PROGRAM MAIN
VAR_OUTPUT
	localTime : TIMESTRUCT;
END_VAR
VAR
	execute AT %I* : BOOL;
	trigger : R_TRIG;
	
	newBundle AT %M* : Bundle;
	newBundleConveyorsOccupied : ARRAY[1..6] OF BOOL;
	bundlesQueue : ARRAY[0..CONSTS.maxQueue] OF Bundle;
	numBundles : INT;
	
	buffers : ARRAY[1..CONSTS.numBuffers] OF IndexedBuffer;
END_VAR
VAR //transfer junctions are clear
	transferJunctionClear_A4 AT %I* : BOOL;
	transferJunctionClear_A5 AT %I* : BOOL;
	transferJunctionClear_A2 AT %I* : BOOL;
END_VAR
VAR CONSTANT //area 3 indexes for the transfer junctions
	transferJunctionIndex_A4 : INT := 5;
	transferJunctionIndex_A5 : INT := 10;
	transferJunctionIndex_A2 : INT := 20;
END_VAR

(*
Area 3 contains <n> buffers, each index contains 6 conveyors
	this allows each buffer to carry up to a theoretical maximum of 6 bundles - realistically this will be limited to 3

implementation:
	each buffer stores 6 iterators (1 for each conveyor) to point to an element in bundlesQueue, and a master conveyor mode request
	set the requested mode for all conveyors within a buffer to the highest priority request
	then use an external module calculate the links and set the modes
	
on receipt of new bundle:
	add to bundle queue
	identify which conveyor lines the bundle sits on
*)

initialize();
callBuffers();

METHOD PRIVATE blocks : BOOL
VAR_INPUT
END_VAR
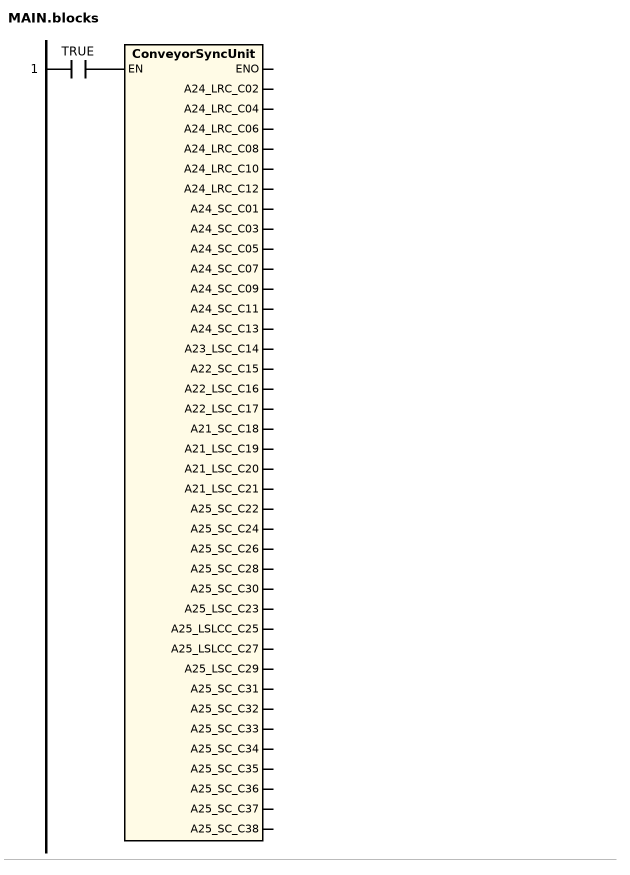
// NETWORK 1
ConveyorSyncUnit();
END_METHOD

METHOD callBuffers : BOOL
VAR_INPUT
END_VAR
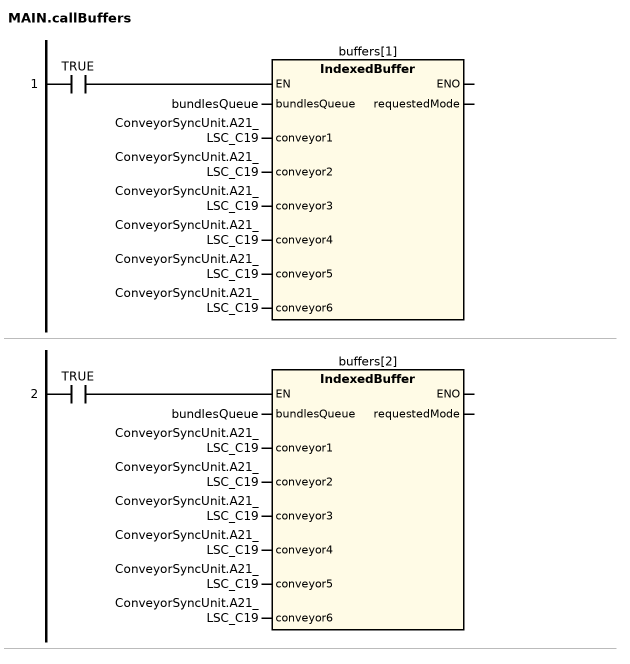
// NETWORK 1
buffers[1](
    bundlesQueue := bundlesQueue,
    conveyor1 := ConveyorSyncUnit.A21_LSC_C19,
    conveyor2 := ConveyorSyncUnit.A21_LSC_C19,
    conveyor3 := ConveyorSyncUnit.A21_LSC_C19,
    conveyor4 := ConveyorSyncUnit.A21_LSC_C19,
    conveyor5 := ConveyorSyncUnit.A21_LSC_C19,
    conveyor6 := ConveyorSyncUnit.A21_LSC_C19); // IndexedBuffer

// NETWORK 2
buffers[2](
    bundlesQueue := bundlesQueue,
    conveyor1 := ConveyorSyncUnit.A21_LSC_C19,
    conveyor2 := ConveyorSyncUnit.A21_LSC_C19,
    conveyor3 := ConveyorSyncUnit.A21_LSC_C19,
    conveyor4 := ConveyorSyncUnit.A21_LSC_C19,
    conveyor5 := ConveyorSyncUnit.A21_LSC_C19,
    conveyor6 := ConveyorSyncUnit.A21_LSC_C19); // IndexedBuffer
END_METHOD

METHOD PRIVATE handleJunctions : BOOL
VAR_INPUT
END_VAR
(*
special junction indexes (temporary):
	A4: 5
	A5: 10
	A2: 20
*)

(*
if junction is occupied:
	conveyor before junction cannot move FWD
	conveyor after junction cannot move BCK
	
consecutive occupied conveyors must be chained to the same motion
	use ConveyorSyncUnit PRG
*)
END_METHOD

METHOD PRIVATE initialize : BOOL
VAR
	i : INT;
END_VAR
FOR i:=1 TO CONSTS.numBuffers-1 BY 1 DO
	buffers[i].connectTo(next:= ADR(buffers[i+1]));
END_FOR
END_METHOD

METHOD PRIVATE receive : BOOL
VAR
	i : DINT;
END_VAR
FOR i:=0 TO CONSTS.maxQueue BY 1 DO
	
	IF NOT BundleIsValid(bundlesQueue[i]) THEN
		bundlesQueue[i] := newBundle;
		
		receive := TRUE;
		EXIT;
	END_IF
	
END_FOR

//read newBundleConveyorsOccupied[] to see which conveyor lines the bundle sits on
END_METHOD

END_PROGRAM

(* stored: Version 1.1.0.1, ProductVersion 3.1.4024.11
   POU MAIN: Id {b937086c-4ebe-4a76-ae0c-99b670c8de9b}, SpecialFunc None
   Method blocks: Id {dbc7b1c8-ae30-41be-9c21-5e864432003b}
   Method callBuffers: Id {f341e8b2-6a00-4e29-bcc3-385c1c378dc5}
   Method handleJunctions: Id {b64f4e2b-a6e8-45e4-b980-f01202879ead}
   Method initialize: Id {19369dbe-d3cd-436d-bd29-dcce27157f3e}
   Method receive: Id {afd27d4a-372a-47c4-8d0e-133fd776335d} *)
